TYPE E_ConveyorState :
(
    Idle := 0,
    Starting,
    Running,
    Fault
);
END_TYPE

(* stored: Version 1.1.0.1, ProductVersion 3.1.4024.12
   DUT E_ConveyorState: Id {a1b2c3d4-0020-4000-8000-000000000020} *)
